FUNCTION_BLOCK T_GetHandle EXTENDS T_NamedBase IMPLEMENTS I_TaskState;
VAR
   _symbolHandle : REFERENCE TO ST_SymbolHandle; // just for debug
   readWrite : T_AdsReadWrite;

END_VAR
VAR CONSTANT
   NO_ERR : UDINT := 0;
   LOG_DEBUG : DWORD := 0;
   LOG_INFO : DWORD := ADSLOG_MSGTYPE_HINT;
   LOG_WARNING : DWORD := ADSLOG_MSGTYPE_WARN;
   LOG_ERROR : DWORD := ADSLOG_MSGTYPE_ERROR;
END_VAR

readWrite();

PROPERTY Busy : BOOL
GET
Busy := readWrite.Busy;
END_GET
END_PROPERTY

PROPERTY Done : BOOL
GET
Done := readWrite.Done;
END_GET
END_PROPERTY

PROPERTY Error : BOOL
GET
Error := readWrite.Error;
END_GET
END_PROPERTY

METHOD TryGetHandle : BOOL
VAR_IN_OUT
   symbolHandle : ST_SymbolHandle; // This handle object will be used in the next step.
END_VAR
VAR_INPUT
   adsTimeout : TIME := DEFAULT_ADS_TIMEOUT; // DEFAULT_ADS_TIMEOUT is T#5s;
END_VAR
VAR_OUTPUT
   status : I_TaskState;
END_VAR
VAR
   readWriteOpts : ST_AdsReadWriteOptions;
END_VAR
VAR CONSTANT
   NO_HANDLE : DWORD := 0;
END_VAR
IF Busy THEN
   LogWarning('Cannot TryGetHandle as Busy');
   RETURN;

END_IF

_symbolHandle REF= symbolHandle;

readWriteOpts.AdsAddress := symbolHandle.SymbolAddress.Ads;
readWriteOpts.IndexGroup := ADSIGRP_SYM_HNDBYNAME;
readWriteOpts.IndexOffset := 0;
readWriteOpts.WriteParams := F_STRING(symbolHandle.SymbolAddress.SymbolName);
readWriteOpts.ReadParams := F_DWORD(symbolHandle.Handle);
readWriteOpts.Timeout := adsTimeout;

TryGetHandle := readWrite.TryRequest(readWriteOpts, status => status);
END_METHOD

END_FUNCTION_BLOCK

(* stored: Version 1.1.0.1, ProductVersion 3.1.4024.9
   POU T_GetHandle: Id {0d283210-5f29-4d37-a1f8-b0443bbf3140}, SpecialFunc None
   Property Busy: Id {9d17c277-f4c0-4a0d-a4a5-2cccea81f8f9}
   Get Get: Id {94da8554-c43e-4933-b298-0bcaf6a8f017}
   Property Done: Id {5af1623b-569a-47e2-84b0-d7d735fea09b}
   Get Get: Id {e9eaa185-d403-41c4-b5e5-7712c4acb10f}
   Property Error: Id {70bba137-79e2-44be-a2b8-680575174dc1}
   Get Get: Id {f2f887f6-2f23-4461-814d-3ebbdfaeeaa7}
   Method TryGetHandle: Id {27b2eda7-b141-42d9-96ab-bdcec3e2ab6a} *)
